// TIA Portal V15.1 export
// export: Created 2026-01-09T13:45:11.4773517Z, ExportSetting WithDefaults, WithReadOnly, DisplayName Totally Integrated Automation Portal, DisplayVersion V15.1 Update 8, DisplayName TIA Portal Openness, DisplayVersion V15.1 Update 8, DisplayName STEP 7 Professional, DisplayVersion V15.1 Update 8, DisplayName WinCC Advanced, DisplayVersion V15.1 Update 8
DATA_BLOCK "C#1_RB"   // DB1
{ S7_Optimized_Access := 'FALSE' }
VERSION : 0.1
// stored: AutoNumber true, CodeModifiedDate 2024-10-21T16:21:19.3207346Z, CompileDate 2025-08-30T17:40:33.1183285Z, CreationDate 2024-10-12T12:36:08.0193576Z, DBAccessibleFromOPCUA true, InterfaceModifiedDate 2024-10-21T16:21:19.3207346Z, IsConsistent true, IsKnowHowProtected false, IsOnlyStoredInLoadMemory false, IsPLCDB false, IsWriteProtectedInAS false, ModifiedDate 2024-10-21T16:21:19.3207346Z, ParameterModified 2024-10-21T16:21:19.3207346Z, StructureModified 2024-10-21T16:21:19.3207346Z
   VAR
      "TH. NOI TRON" : Bool;   // Tín hiệu nồi trộn
      "TH. BTX" : Bool;   // Tín hiệu băng tải xiên
      "TH. BTN" : Bool;   // Tín hiệu băng tải ngang
      "TH. TANG SAY" : Bool;   // Tín hiệu tang sấy cốt liệu
      "TH. GAU COT LIEU" : Bool;   // Tín hiệu gàu tải cốt liệu nóng
      "TH. GAU F/D" : Bool;   // Tín hiệu gàu tải phụ gia bột
      "TH. SAN RUNG" : Bool;   // Tín hiệu sàng rung cốt liệu nóng
      "TH. CUA DONG" : Bool;   // Tín hiệu cửa nồi trộn đóng
      "TH. CUA MO" : Bool;   // Tín hiệu cửa nồi trộn mở
      "TH. MNK" : Bool;   // Tín hiệu máy nén khí chạy
      "TH. TRAN AG1" : Bool;   // Tín hiệu báo tràn silo AG1
      "TH. TRAN AG2" : Bool;   // Tín hiệu báo tràn silo AG2
      "TH. TRAN AG3" : Bool;   // Tín hiệu báo tràn silo AG3
      "TH. TRAN AG4" : Bool;   // Tín hiệu báo tràn silo AG4
      "TH. TRAN AG5" : Bool;   // Tín hiệu báo tràn silo AG5
      "TH. TRAN FD1" : Bool;   // Tín hiệu báo tràn silo F/D
      "TH. TRAN SB1" : Bool;   // Tín hiệu báo tràn silo SBS
      "TH. SILO FD HIGHT" : Bool;   // Tín hiệu báo mức cao silo chứa F/D
      "TH. SILO FD LOW" : Bool;   // Tín hiệu báo mức thấp silo chứa F/D
      "NOI TRON" : Bool;   // Nồi trộn
      BTX : Bool;   // Băng tải xiên
      BTN : Bool;   // Băng tải ngang
      "TANG SAY" : Bool;   // Tang sấy cốt liệu
      "BOM DAU" : Bool;   // Bơm dầu DO
      "GAU COT LIEU" : Bool;   // Gàu tải cốt liệu nóng
      "SAN RUNG" : Bool;   // Sàn rung cốt liệu
      "GAU FD" : Bool;   // Gàu tải phụ F/D
      "VIT TAI FD" : Bool;   // Vít tải F/D
      "BOM SBS" : Bool;   // Bơm nạp hạt nhựa SBS
      "QUAT GIO" : Bool;   // Quạt gió lọc bụi
      "BOM NUOC" : Bool;   // Bơm nước lọc bụi
      "MO CUA" : Bool;   // Van mở cửa nồi trộn
      "DONG CUA" : Bool;   // Van đóng cửa nồi trộn
      MNK : Bool;   // Máy nén khí
      "XA CL1" : Bool;   // Băng tải xả cốt liệu 1
      "XA CL2" : Bool;   // Băng tải xả cốt liệu 2
      "XA CL3" : Bool;   // Băng tải xả cốt liệu 3
      "XA CL4" : Bool;   // Băng tải xả cốt liệu 4
      "XA CL5" : Bool;   // Băng tải xả cốt liệu 5
      "CAN AG1" : Bool;   // Van cân AG1
      "CAN AG2" : Bool;   // Van cân AG2
      "CAN AG3" : Bool;   // Van cân AG3
      "CAN AG4" : Bool;   // Van cân AG4
      "CAN AG5" : Bool;   // Van cân AG5
      "CAN FD1" : Bool;   // Van cân F/D
      "CAN AP1" : Bool;   // Bơm nhựa
      "CAN SB1" : Bool;   // Van cân hạt nhựa SBS
      "XA W_AG1" : Bool;   // Van xả cân AG1
      "XA W_FD1" : Bool;   // Van xả cân FD1
      "XA W_AP1" : Bool;   // Van xả cân AP1
      "XA W_SB1" : Bool;   // Van xả cân SB1
      BOM_TUOI_NHUA : Bool;   // Bổ sung 1
      DAU_DOT : Bool;   // Bổ sung 2
      VAN_PNSBS : Bool;   // Bổ sung 3
      "RUNG CL1" : Bool;   // Bổ sung 4
      "RUNG CL2" : Bool;   // Bổ sung 5
      "RUNG CL3" : Bool;   // Bổ sung 6
      "NOTE 7" : Bool;   // Bổ sung 7
      RUNNING : Bool;   // Trạng thái đang trộn
      SIMULATION : Bool;   // Trạng thái chạy mô phỏng
      MIXER_FULL : Bool;   // Trạng thái nồi trộn báo đầy
      TTC_AG1 : Bool;   // Trạng thái cân Ag1
      TTC_AG2 : Bool;   // Trạng thái cân Ag2
      TTC_AG3 : Bool;   // Trạng thái cân Ag3
      TTC_AG4 : Bool;   // Trạng thái cân Ag4
      TTC_AG5 : Bool;   // Trạng thái cân Ag5
      TTC_FD1 : Bool;   // Trạng thái cân FD1
      TTC_AP1 : Bool;   // Trạng thái cân AP1
      TTC_SB1 : Bool;   // Trạng thái cân SBS1
   END_VAR
BEGIN
END_DATA_BLOCK
